(* CoDeSys 2.3 export: CHECKDIVBYTE.EXP *)

(* POU CheckDivByte, ST *)
FUNCTION CheckDivByte : BYTE
VAR_INPUT
	divisor: BYTE;
END_VAR
VAR
END_VAR
(* @TEXT_IMPLEMENTATION := 'ST' *)
IF divisor = 0 THEN
	CheckDivByte := 1;
ELSE
	CheckDivByte := divisor;
END_IF
END_FUNCTION
